FUNCTION_BLOCK PUBLIC PAEEMotorFreq1D EXTENDS PAEEMotorFreqCtrl
VAR_INPUT
END_VAR
VAR_OUTPUT
END_VAR
VAR
	_PAPointMatIn1 : PAPoint(THIS^);
	_PAPointMatOut1 : PAPoint(THIS^);
END_VAR

METHOD FB_init : BOOL
VAR_INPUT
	bInitRetains : BOOL; // if TRUE, the retain variables are initialized (warm start / cold start)
	bInCopyCode : BOOL;  // if TRUE, the instance afterwards gets moved into the copy code (online change)
	parent : IACComponent;
END_VAR
AddPoint(_PAPointMatIn1);
AddPoint(_PAPointMatOut1);
END_METHOD

METHOD PUBLIC HasPointReachedOffPosition : BOOL
VAR_INPUT
	point : IACPoint;
END_VAR
IF point = PAPointMatOut1 THEN
	HasPointReachedOffPosition := NOT _RunState;
ELSIF point = PAPointMatIn1 THEN
	HasPointReachedOffPosition := TRUE;
ELSE
	HasPointReachedOffPosition := FALSE;
END_IF
END_METHOD

METHOD PUBLIC HasPointReachedOnPosition : BOOL
VAR_INPUT
	point : IACPoint;
END_VAR
IF point = PAPointMatOut1 THEN
	HasPointReachedOnPosition :=     _RunState
								AND (   (_Speed >= (_ReqSpeed - 0.001))
									 OR (_Speed >= (_DesiredSpeed - 0.001)));
ELSIF point = PAPointMatIn1 THEN
	HasPointReachedOnPosition := TRUE;
ELSE
	HasPointReachedOnPosition := FALSE;
END_IF
END_METHOD

METHOD PUBLIC IsEnabledTurnOn : BOOL
VAR_INPUT
END_VAR
END_METHOD

PROPERTY PUBLIC PAPointMatIn1 : IACPoint
GET // PUBLIC
PAPointMatIn1 := _PAPointMatIn1;
END_GET
END_PROPERTY

PROPERTY PUBLIC PAPointMatOut1 : IACPoint
GET // PUBLIC
PAPointMatOut1 := _PAPointMatOut1;
END_GET
END_PROPERTY

METHOD PUBLIC TurnOn
VAR_INPUT
END_VAR
END_METHOD

METHOD PUBLIC TurnOnWithSpeed
VAR_INPUT
END_VAR
END_METHOD

END_FUNCTION_BLOCK

(* stored: Version 1.1.0.1, ProductVersion 3.1.4020.12
   POU PAEEMotorFreq1D: Id {ae4507dd-07d2-44e5-b4ca-69bd88ebd543}, SpecialFunc None
   Method FB_init: Id {f242c4f6-3e98-4d16-9307-c60e6ec269cb}
   Method HasPointReachedOffPosition: Id {ae9111ac-b041-4788-bf67-42623f2e1d3e}
   Method HasPointReachedOnPosition: Id {4a6f5f17-040a-44cc-93d4-29a9d0f08092}
   Method IsEnabledTurnOn: Id {3957f70c-c352-4cfd-bf9c-4fafa51fab65}
   Property PAPointMatIn1: Id {071cfea4-0168-475a-9e75-15b4ddc395df}
   Get Get: Id {9d23a74b-dbae-4ebc-b985-487313104442}
   Property PAPointMatOut1: Id {0d1cfbf1-ff75-4933-bec0-a02615963bbe}
   Get Get: Id {90babcd4-3a90-4691-825a-e0e4b6061672}
   Method TurnOn: Id {9c3382a7-df2e-4fd8-9726-ceb73d1e069a}
   Method TurnOnWithSpeed: Id {d3d61397-ba3f-498f-af57-86920ec06872} *)
